{attribute 'qualified_only'} // optional: forces qualified access with GVL_B.
VAR_GLOBAL
    rTemperature : REAL := 75.5;
    bAlarm       : BOOL := FALSE;
    bAckFromA    : BOOL := FALSE;   // Project A writes TRUE here
END_VAR

(* stored: Version 1.1.0.1, ProductVersion 3.1.4024.16
   GVL GVL_B: Id {83978245-e4f7-47f0-9d75-fa2497095eda} *)
